# EPICS substitutions: ioc/bsreadtest.subs
file bsreadtest.template {
	pattern{P} {BSREAD-TEST}
}
